(* Logix 5000 project; controller Amvex_Thorpe_Flowmeter vendor 1 type 14 code 106 rev 33.13; software revision 33.01; part 11 of 16 *)
(* tags used below, declared in another part *)
   Auto_Seq : SEQ;
   Manual_ONS : BOOL;
   Manual_Output_Reset : BOOL;
   MODE : MODE;
   RESET : BOOL;
   temp_Gripper_Delay : TIMER;
   Test : Connect;
   Air_Pressure_Issue_Delay_TMR : TIMER;
   Close : BOOL;
   Close_Rapid : Servo_Move;
   Close_Step : Servo_Move;
   Datalogging_Time_Delay : TIMER;
   HMI : HMI_Temp;
   MCP : MCP;
   MCP_00 : UDT_ID86;
   Open : BOOL;
   Reject : BOOL;
   Reject_Active : BOOL;
   Reject_Pallet_Bit : DINT;
   Test2_Step : Servo_Move;
   Test4_Step : Servo_Move;
   Test5_Step : Servo_Move;
   Test_Data : REAL[8];
   Test_Data_ONS : BOOL[32];
   Test_Delay_TMR : TIMER[5];
   Transmit_Data : BOOL;
   Vision_Result_OK_TMR : TIMER[6];
   Vision_TMR : TIMER[3];
(* MCP_Main, continued *)

ROUTINE NEW_YEAR   (* ladder *)
END_ROUTINE

ROUTINE R01_INPUTS   (* ladder *)
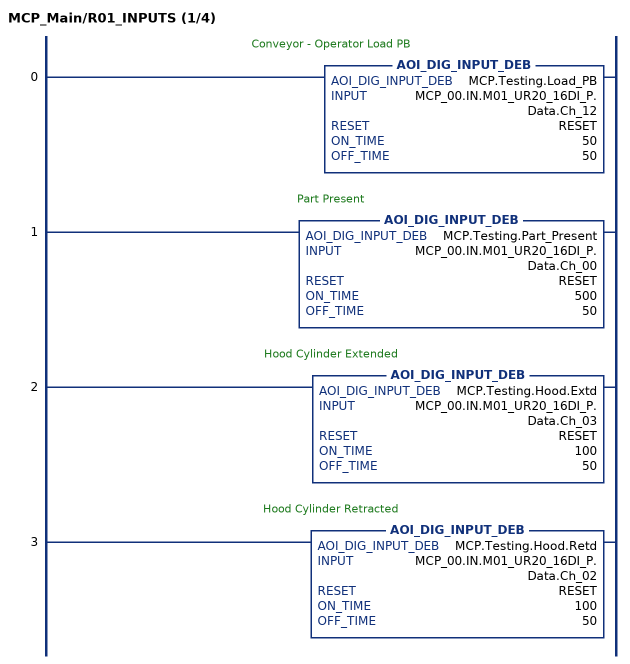
   // Conveyor - Operator Load PB
   0: AOI_DIG_INPUT_DEB(MCP.Testing.Load_PB,MCP_00.IN.M01_UR20_16DI_P.Data.Ch_12,RESET,50,50);
   // Part Present
   1: AOI_DIG_INPUT_DEB(MCP.Testing.Part_Present,MCP_00.IN.M01_UR20_16DI_P.Data.Ch_00,RESET,500,50);
   // Hood Cylinder Extended
   2: AOI_DIG_INPUT_DEB(MCP.Testing.Hood.Extd,MCP_00.IN.M01_UR20_16DI_P.Data.Ch_03,RESET,100,50);
   // Hood Cylinder Retracted
   3: AOI_DIG_INPUT_DEB(MCP.Testing.Hood.Retd,MCP_00.IN.M01_UR20_16DI_P.Data.Ch_02,RESET,100,50);
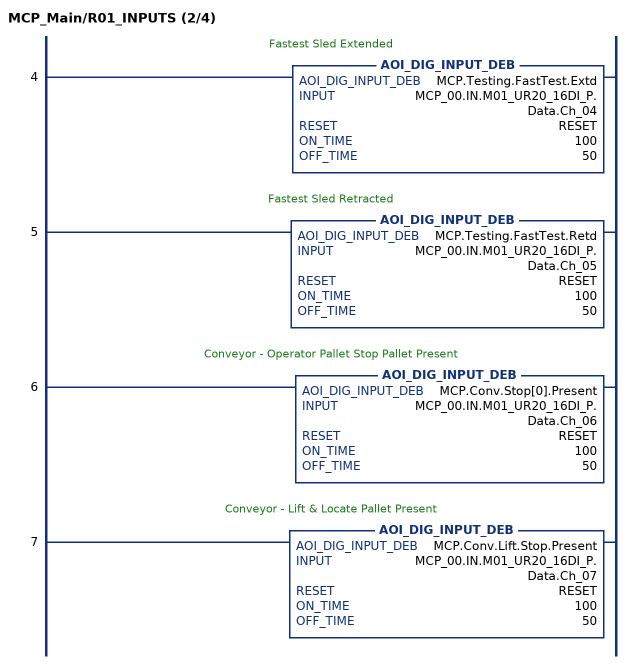
   // Fastest Sled Extended
   4: AOI_DIG_INPUT_DEB(MCP.Testing.FastTest.Extd,MCP_00.IN.M01_UR20_16DI_P.Data.Ch_04,RESET,100,50);
   // Fastest Sled Retracted
   5: AOI_DIG_INPUT_DEB(MCP.Testing.FastTest.Retd,MCP_00.IN.M01_UR20_16DI_P.Data.Ch_05,RESET,100,50);
   // Conveyor - Operator Pallet Stop Pallet Present
   6: AOI_DIG_INPUT_DEB(MCP.Conv.Stop[0].Present,MCP_00.IN.M01_UR20_16DI_P.Data.Ch_06,RESET,100,50);
   // Conveyor - Lift & Locate Pallet Present
   7: AOI_DIG_INPUT_DEB(MCP.Conv.Lift.Stop.Present,MCP_00.IN.M01_UR20_16DI_P.Data.Ch_07,RESET,100,50);
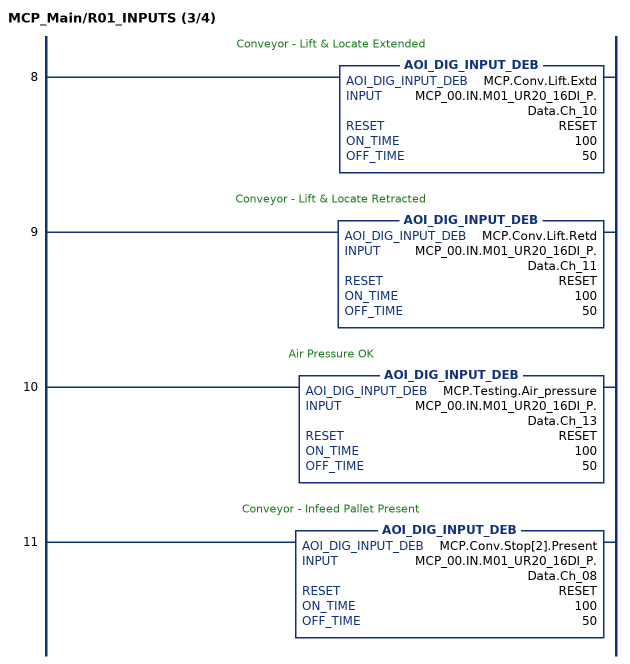
   // Conveyor - Lift & Locate Extended
   8: AOI_DIG_INPUT_DEB(MCP.Conv.Lift.Extd,MCP_00.IN.M01_UR20_16DI_P.Data.Ch_10,RESET,100,50);
   // Conveyor - Lift & Locate Retracted
   9: AOI_DIG_INPUT_DEB(MCP.Conv.Lift.Retd,MCP_00.IN.M01_UR20_16DI_P.Data.Ch_11,RESET,100,50);
   // Air Pressure OK
   10: AOI_DIG_INPUT_DEB(MCP.Testing.Air_pressure,MCP_00.IN.M01_UR20_16DI_P.Data.Ch_13,RESET,100,50);
   // Conveyor - Infeed Pallet Present
   11: AOI_DIG_INPUT_DEB(MCP.Conv.Stop[2].Present,MCP_00.IN.M01_UR20_16DI_P.Data.Ch_08,RESET,100,50);
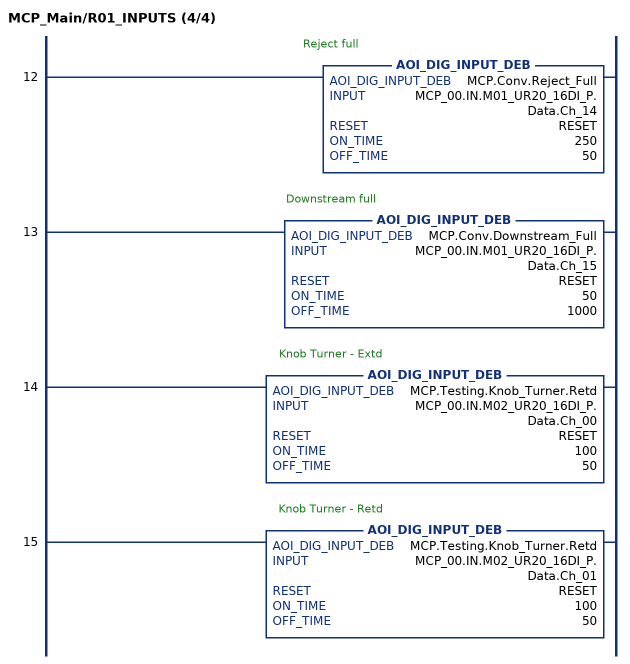
   // Reject full
   12: AOI_DIG_INPUT_DEB(MCP.Conv.Reject_Full,MCP_00.IN.M01_UR20_16DI_P.Data.Ch_14,RESET,250,50);
   // Downstream full
   13: AOI_DIG_INPUT_DEB(MCP.Conv.Downstream_Full,MCP_00.IN.M01_UR20_16DI_P.Data.Ch_15,RESET,50,1000);
   // Knob Turner - Extd
   14: AOI_DIG_INPUT_DEB(MCP.Testing.Knob_Turner.Retd,MCP_00.IN.M02_UR20_16DI_P.Data.Ch_00,RESET,100,50);
   // Knob Turner - Retd
   15: AOI_DIG_INPUT_DEB(MCP.Testing.Knob_Turner.Retd,MCP_00.IN.M02_UR20_16DI_P.Data.Ch_01,RESET,100,50);
END_ROUTINE

ROUTINE R02_OUTPUTS   (* ladder *)
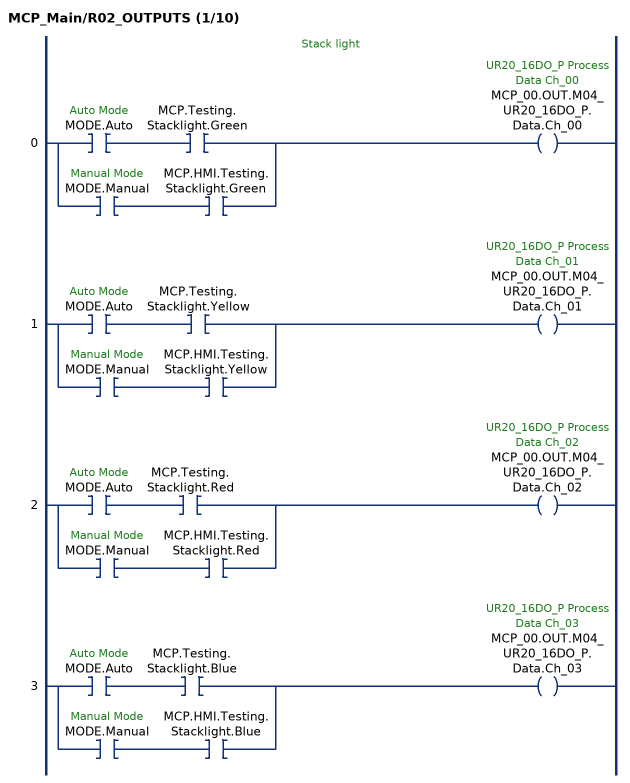
   // Stack light
   0: [XIC(MODE.Auto) XIC(MCP.Testing.Stacklight.Green) ,XIC(MODE.Manual) XIC(MCP.HMI.Testing.Stacklight.Green) ]OTE(MCP_00.OUT.M04_UR20_16DO_P.Data.Ch_00);
   1: [XIC(MODE.Auto) XIC(MCP.Testing.Stacklight.Yellow) ,XIC(MODE.Manual) XIC(MCP.HMI.Testing.Stacklight.Yellow) ]OTE(MCP_00.OUT.M04_UR20_16DO_P.Data.Ch_01);
   2: [XIC(MODE.Auto) XIC(MCP.Testing.Stacklight.Red) ,XIC(MODE.Manual) XIC(MCP.HMI.Testing.Stacklight.Red) ]OTE(MCP_00.OUT.M04_UR20_16DO_P.Data.Ch_02);
   3: [XIC(MODE.Auto) XIC(MCP.Testing.Stacklight.Blue) ,XIC(MODE.Manual) XIC(MCP.HMI.Testing.Stacklight.Blue) ]OTE(MCP_00.OUT.M04_UR20_16DO_P.Data.Ch_03);
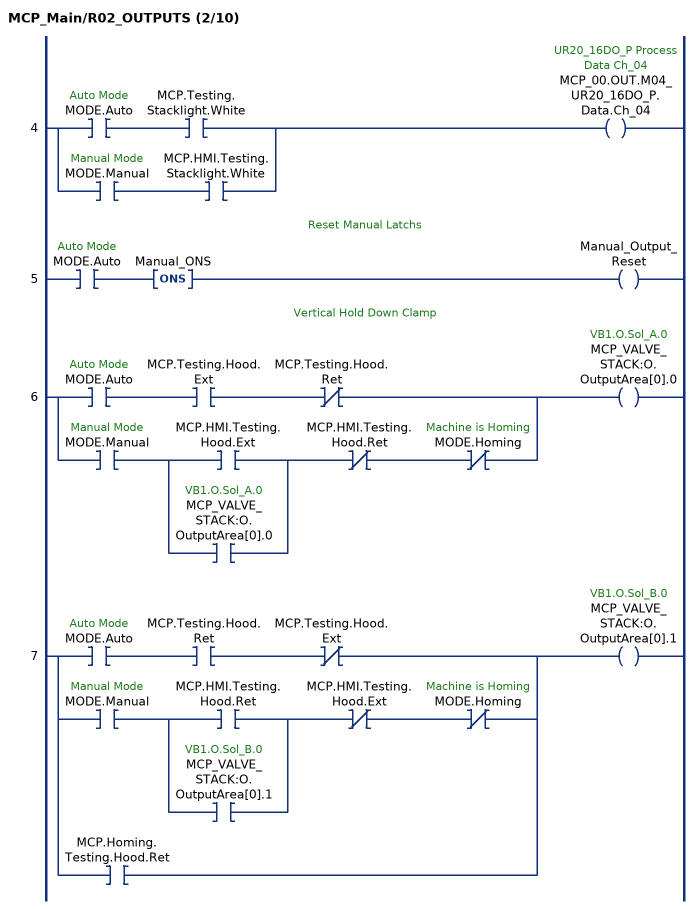
   4: [XIC(MODE.Auto) XIC(MCP.Testing.Stacklight.White) ,XIC(MODE.Manual) XIC(MCP.HMI.Testing.Stacklight.White) ]OTE(MCP_00.OUT.M04_UR20_16DO_P.Data.Ch_04);
   // Reset Manual Latchs
   5: XIC(MODE.Auto)ONS(Manual_ONS)OTE(Manual_Output_Reset);
   // Vertical Hold Down Clamp
   6: [XIC(MODE.Auto) XIC(MCP.Testing.Hood.Ext) XIO(MCP.Testing.Hood.Ret) ,XIC(MODE.Manual) [XIC(MCP.HMI.Testing.Hood.Ext) ,XIC(MCP_VALVE_STACK:O.OutputArea[0].0) ] XIO(MCP.HMI.Testing.Hood.Ret) XIO(MODE.Homing) ]OTE(MCP_VALVE_STACK:O.OutputArea[0].0);
   7: [XIC(MODE.Auto) XIC(MCP.Testing.Hood.Ret) XIO(MCP.Testing.Hood.Ext) ,XIC(MODE.Manual) [XIC(MCP.HMI.Testing.Hood.Ret) ,XIC(MCP_VALVE_STACK:O.OutputArea[0].1) ] XIO(MCP.HMI.Testing.Hood.Ext) XIO(MODE.Homing) ,XIC(MCP.Homing.Testing.Hood.Ret) ]OTE(MCP_VALVE_STACK:O.OutputArea[0].1);
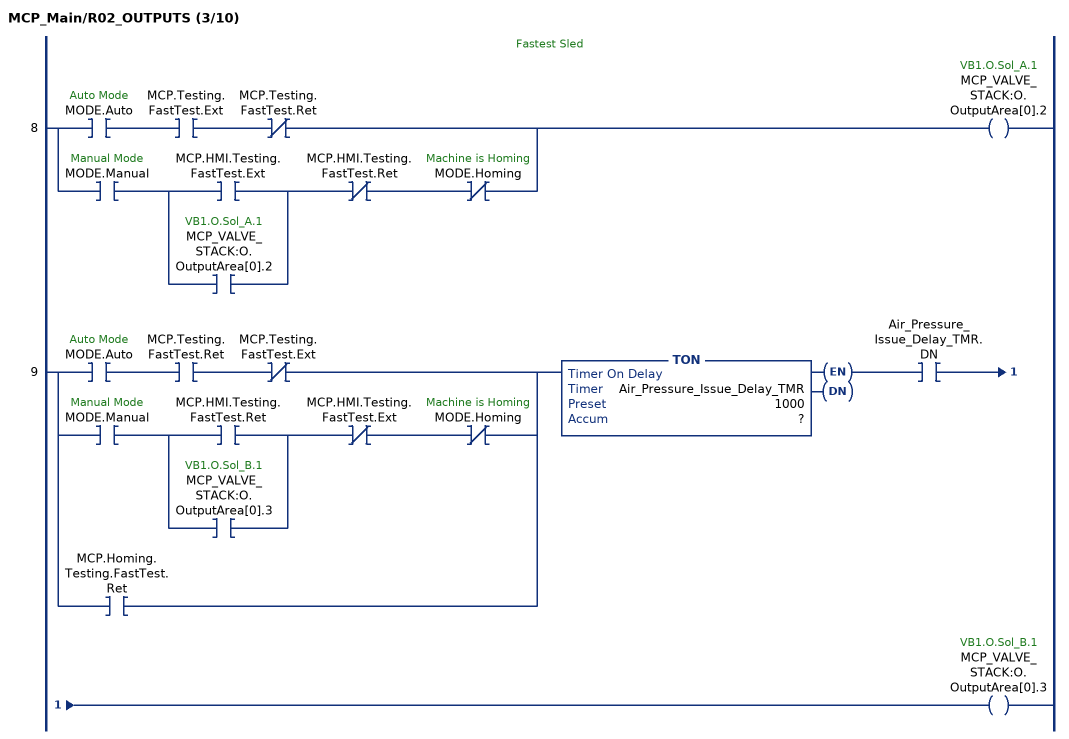
   // Fastest Sled
   8: [XIC(MODE.Auto) XIC(MCP.Testing.FastTest.Ext) XIO(MCP.Testing.FastTest.Ret) ,XIC(MODE.Manual) [XIC(MCP.HMI.Testing.FastTest.Ext) ,XIC(MCP_VALVE_STACK:O.OutputArea[0].2) ] XIO(MCP.HMI.Testing.FastTest.Ret) XIO(MODE.Homing) ]OTE(MCP_VALVE_STACK:O.OutputArea[0].2);
   9: [XIC(MODE.Auto) XIC(MCP.Testing.FastTest.Ret) XIO(MCP.Testing.FastTest.Ext) ,XIC(MODE.Manual) [XIC(MCP.HMI.Testing.FastTest.Ret) ,XIC(MCP_VALVE_STACK:O.OutputArea[0].3) ] XIO(MCP.HMI.Testing.FastTest.Ext) XIO(MODE.Homing) ,XIC(MCP.Homing.Testing.FastTest.Ret) ]TON(Air_Pressure_Issue_Delay_TMR,?,?)XIC(Air_Pressure_Issue_Delay_TMR.DN)OTE(MCP_VALVE_STACK:O.OutputArea[0].3);
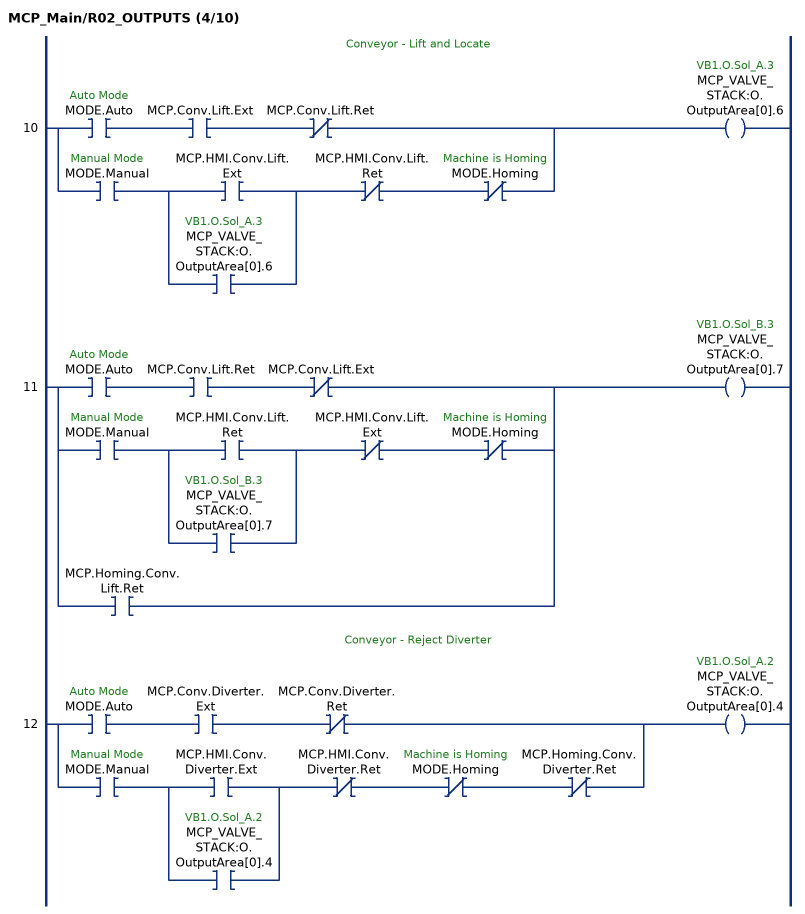
   // Conveyor - Lift and Locate
   10: [XIC(MODE.Auto) XIC(MCP.Conv.Lift.Ext) XIO(MCP.Conv.Lift.Ret) ,XIC(MODE.Manual) [XIC(MCP.HMI.Conv.Lift.Ext) ,XIC(MCP_VALVE_STACK:O.OutputArea[0].6) ] XIO(MCP.HMI.Conv.Lift.Ret) XIO(MODE.Homing) ]OTE(MCP_VALVE_STACK:O.OutputArea[0].6);
   11: [XIC(MODE.Auto) XIC(MCP.Conv.Lift.Ret) XIO(MCP.Conv.Lift.Ext) ,XIC(MODE.Manual) [XIC(MCP.HMI.Conv.Lift.Ret) ,XIC(MCP_VALVE_STACK:O.OutputArea[0].7) ] XIO(MCP.HMI.Conv.Lift.Ext) XIO(MODE.Homing) ,XIC(MCP.Homing.Conv.Lift.Ret) ]OTE(MCP_VALVE_STACK:O.OutputArea[0].7);
   // Conveyor - Reject Diverter
   12: [XIC(MODE.Auto) XIC(MCP.Conv.Diverter.Ext) XIO(MCP.Conv.Diverter.Ret) ,XIC(MODE.Manual) [XIC(MCP.HMI.Conv.Diverter.Ext) ,XIC(MCP_VALVE_STACK:O.OutputArea[0].4) ] XIO(MCP.HMI.Conv.Diverter.Ret) XIO(MODE.Homing) XIO(MCP.Homing.Conv.Diverter.Ret) ]OTE(MCP_VALVE_STACK:O.OutputArea[0].4);
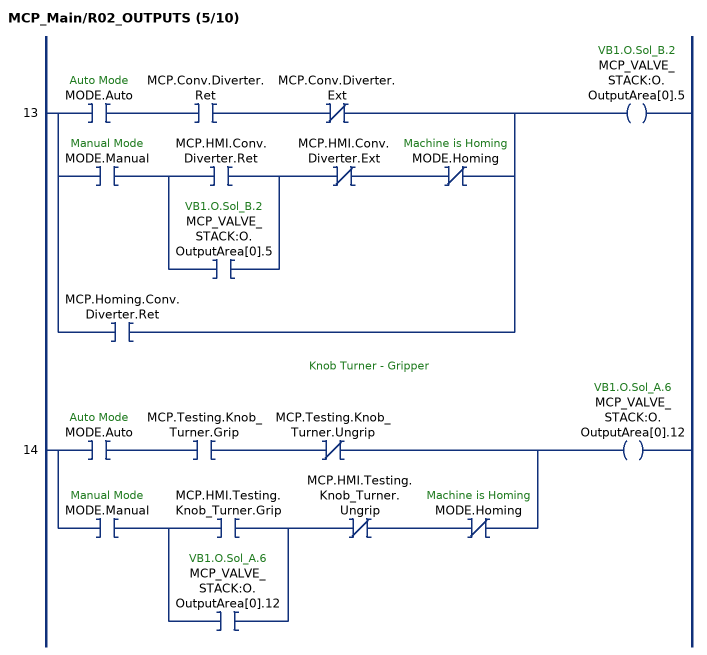
   13: [XIC(MODE.Auto) XIC(MCP.Conv.Diverter.Ret) XIO(MCP.Conv.Diverter.Ext) ,XIC(MODE.Manual) [XIC(MCP.HMI.Conv.Diverter.Ret) ,XIC(MCP_VALVE_STACK:O.OutputArea[0].5) ] XIO(MCP.HMI.Conv.Diverter.Ext) XIO(MODE.Homing) ,XIC(MCP.Homing.Conv.Diverter.Ret) ]OTE(MCP_VALVE_STACK:O.OutputArea[0].5);
   // Knob Turner - Gripper
   14: [XIC(MODE.Auto) XIC(MCP.Testing.Knob_Turner.Grip) XIO(MCP.Testing.Knob_Turner.Ungrip) ,XIC(MODE.Manual) [XIC(MCP.HMI.Testing.Knob_Turner.Grip) ,XIC(MCP_VALVE_STACK:O.OutputArea[0].12) ] XIO(MCP.HMI.Testing.Knob_Turner.Ungrip) XIO(MODE.Homing) ]OTE(MCP_VALVE_STACK:O.OutputArea[0].12);
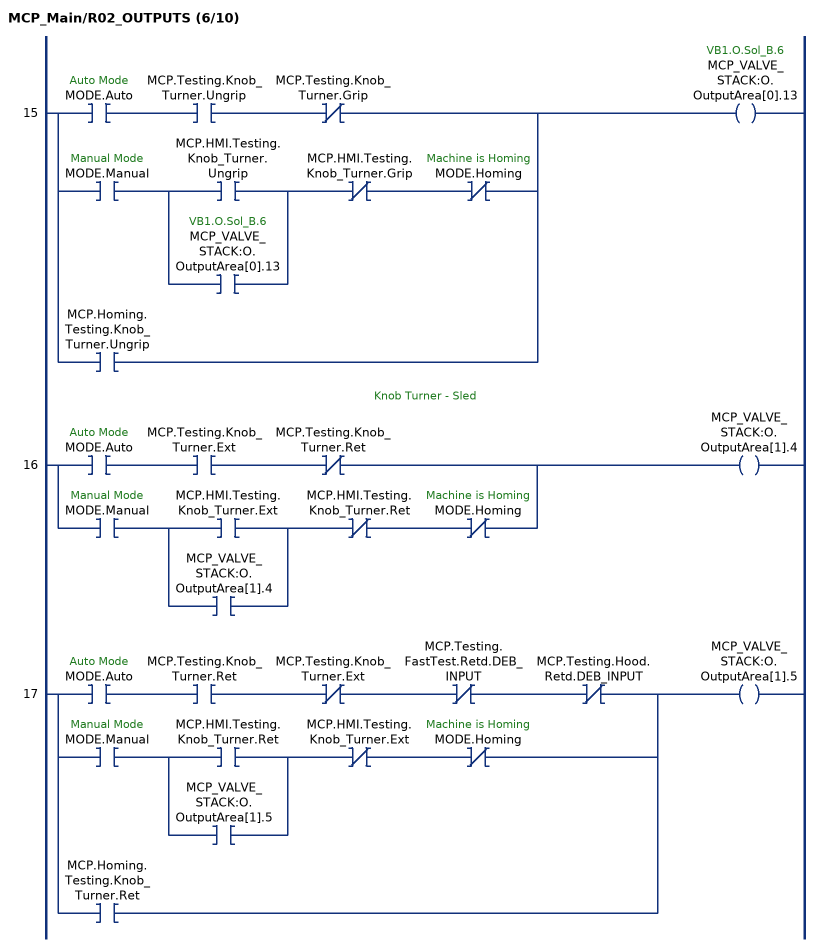
   15: [XIC(MODE.Auto) XIC(MCP.Testing.Knob_Turner.Ungrip) XIO(MCP.Testing.Knob_Turner.Grip) ,XIC(MODE.Manual) [XIC(MCP.HMI.Testing.Knob_Turner.Ungrip) ,XIC(MCP_VALVE_STACK:O.OutputArea[0].13) ] XIO(MCP.HMI.Testing.Knob_Turner.Grip) XIO(MODE.Homing) ,XIC(MCP.Homing.Testing.Knob_Turner.Ungrip) ]OTE(MCP_VALVE_STACK:O.OutputArea[0].13);
   // Knob Turner - Sled
   16: [XIC(MODE.Auto) XIC(MCP.Testing.Knob_Turner.Ext) XIO(MCP.Testing.Knob_Turner.Ret) ,XIC(MODE.Manual) [XIC(MCP.HMI.Testing.Knob_Turner.Ext) ,XIC(MCP_VALVE_STACK:O.OutputArea[1].4) ] XIO(MCP.HMI.Testing.Knob_Turner.Ret) XIO(MODE.Homing) ]OTE(MCP_VALVE_STACK:O.OutputArea[1].4);
   17: [XIC(MODE.Auto) XIC(MCP.Testing.Knob_Turner.Ret) XIO(MCP.Testing.Knob_Turner.Ext) XIO(MCP.Testing.FastTest.Retd.DEB_INPUT) XIO(MCP.Testing.Hood.Retd.DEB_INPUT) ,XIC(MODE.Manual) [XIC(MCP.HMI.Testing.Knob_Turner.Ret) ,XIC(MCP_VALVE_STACK:O.OutputArea[1].5) ] XIO(MCP.HMI.Testing.Knob_Turner.Ext) XIO(MODE.Homing) ,XIC(MCP.Homing.Testing.Knob_Turner.Ret) ]OTE(MCP_VALVE_STACK:O.OutputArea[1].5);
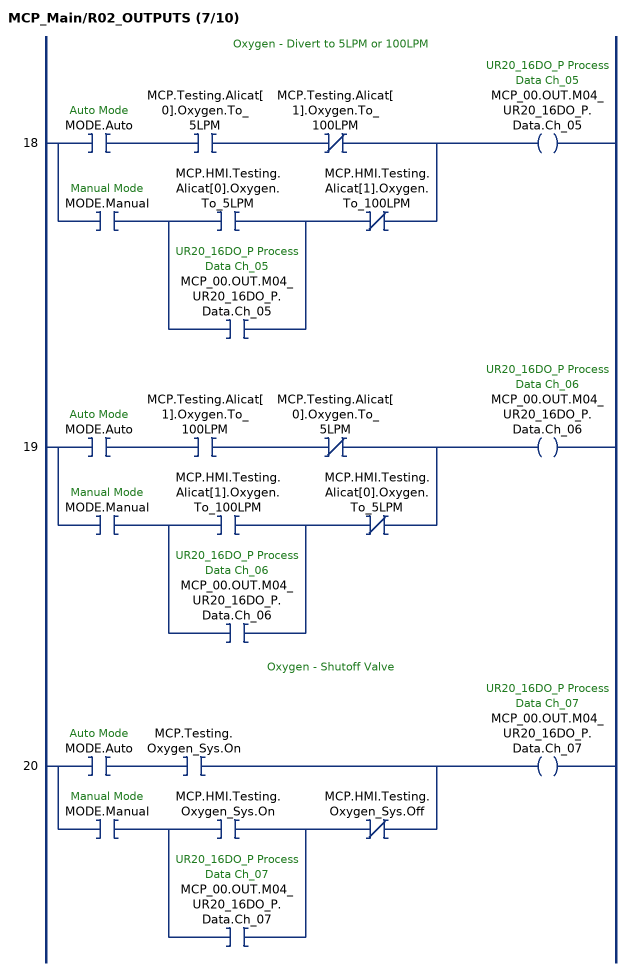
   // Oxygen - Divert to 5LPM or 100LPM
   18: [XIC(MODE.Auto) XIC(MCP.Testing.Alicat[0].Oxygen.To_5LPM) XIO(MCP.Testing.Alicat[1].Oxygen.To_100LPM) ,XIC(MODE.Manual) [XIC(MCP.HMI.Testing.Alicat[0].Oxygen.To_5LPM) ,XIC(MCP_00.OUT.M04_UR20_16DO_P.Data.Ch_05) ] XIO(MCP.HMI.Testing.Alicat[1].Oxygen.To_100LPM) ]OTE(MCP_00.OUT.M04_UR20_16DO_P.Data.Ch_05);
   19: [XIC(MODE.Auto) XIC(MCP.Testing.Alicat[1].Oxygen.To_100LPM) XIO(MCP.Testing.Alicat[0].Oxygen.To_5LPM) ,XIC(MODE.Manual) [XIC(MCP.HMI.Testing.Alicat[1].Oxygen.To_100LPM) ,XIC(MCP_00.OUT.M04_UR20_16DO_P.Data.Ch_06) ] XIO(MCP.HMI.Testing.Alicat[0].Oxygen.To_5LPM) ]OTE(MCP_00.OUT.M04_UR20_16DO_P.Data.Ch_06);
   // Oxygen - Shutoff Valve
   20: [XIC(MODE.Auto) XIC(MCP.Testing.Oxygen_Sys.On) ,XIC(MODE.Manual) [XIC(MCP.HMI.Testing.Oxygen_Sys.On) ,XIC(MCP_00.OUT.M04_UR20_16DO_P.Data.Ch_07) ] XIO(MCP.HMI.Testing.Oxygen_Sys.Off) ]OTE(MCP_00.OUT.M04_UR20_16DO_P.Data.Ch_07);
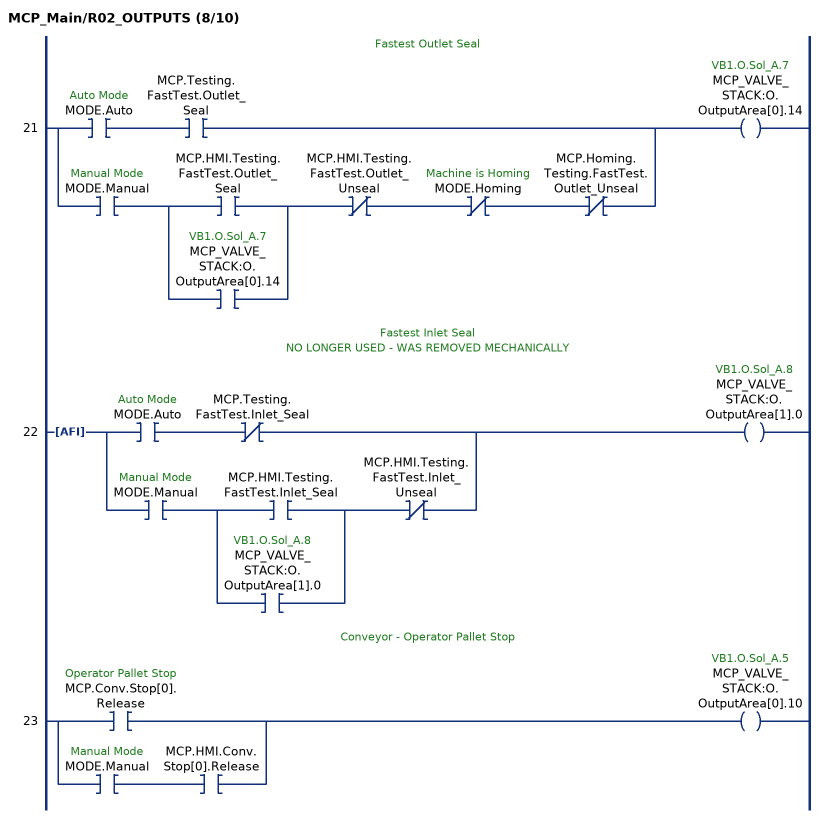
   // Fastest Outlet Seal
   21: [XIC(MODE.Auto) XIC(MCP.Testing.FastTest.Outlet_Seal) ,XIC(MODE.Manual) [XIC(MCP.HMI.Testing.FastTest.Outlet_Seal) ,XIC(MCP_VALVE_STACK:O.OutputArea[0].14) ] XIO(MCP.HMI.Testing.FastTest.Outlet_Unseal) XIO(MODE.Homing) XIO(MCP.Homing.Testing.FastTest.Outlet_Unseal) ]OTE(MCP_VALVE_STACK:O.OutputArea[0].14);
   // Fastest Inlet Seal
   // NO LONGER USED - WAS REMOVED MECHANICALLY
   22: AFI()[XIC(MODE.Auto) XIO(MCP.Testing.FastTest.Inlet_Seal) ,XIC(MODE.Manual) [XIC(MCP.HMI.Testing.FastTest.Inlet_Seal) ,XIC(MCP_VALVE_STACK:O.OutputArea[1].0) ] XIO(MCP.HMI.Testing.FastTest.Inlet_Unseal) ]OTE(MCP_VALVE_STACK:O.OutputArea[1].0);
   // Conveyor - Operator Pallet Stop
   23: [XIC(MCP.Conv.Stop[0].Release) ,XIC(MODE.Manual) XIC(MCP.HMI.Conv.Stop[0].Release) ]OTE(MCP_VALVE_STACK:O.OutputArea[0].10);
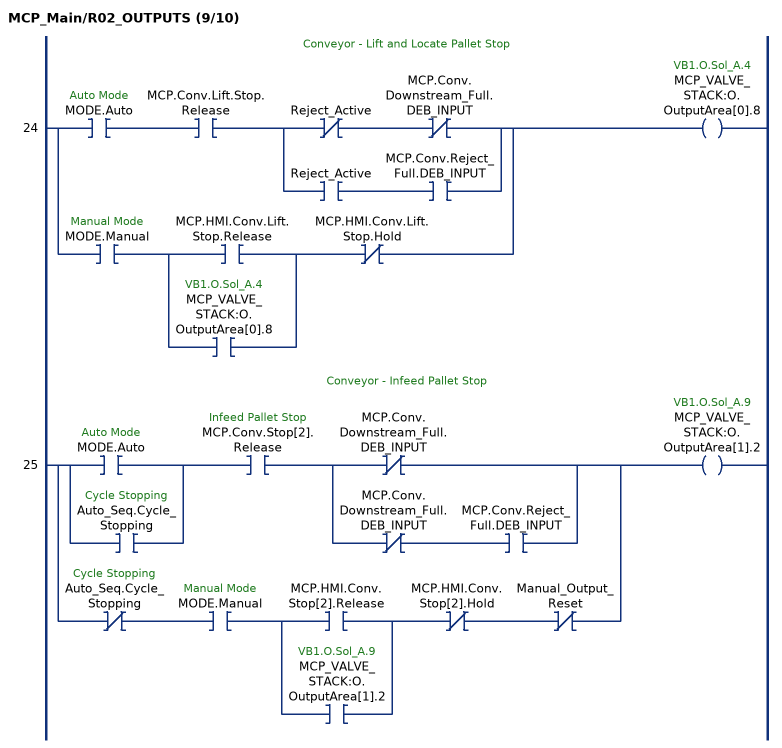
   // Conveyor - Lift and Locate Pallet Stop
   24: [XIC(MODE.Auto) XIC(MCP.Conv.Lift.Stop.Release) [XIO(Reject_Active) XIO(MCP.Conv.Downstream_Full.DEB_INPUT) ,XIC(Reject_Active) XIC(MCP.Conv.Reject_Full.DEB_INPUT) ] ,XIC(MODE.Manual) [XIC(MCP.HMI.Conv.Lift.Stop.Release) ,XIC(MCP_VALVE_STACK:O.OutputArea[0].8) ] XIO(MCP.HMI.Conv.Lift.Stop.Hold) ]OTE(MCP_VALVE_STACK:O.OutputArea[0].8);
   // Conveyor - Infeed Pallet Stop
   25: [[XIC(MODE.Auto) ,XIC(Auto_Seq.Cycle_Stopping) ] XIC(MCP.Conv.Stop[2].Release) [XIO(MCP.Conv.Downstream_Full.DEB_INPUT) ,XIO(MCP.Conv.Downstream_Full.DEB_INPUT) XIC(MCP.Conv.Reject_Full.DEB_INPUT) ] ,XIO(Auto_Seq.Cycle_Stopping) XIC(MODE.Manual) [XIC(MCP.HMI.Conv.Stop[2].Release) ,XIC(MCP_VALVE_STACK:O.OutputArea[1].2) ] XIO(MCP.HMI.Conv.Stop[2].Hold) XIO(Manual_Output_Reset) ]OTE(MCP_VALVE_STACK:O.OutputArea[1].2);
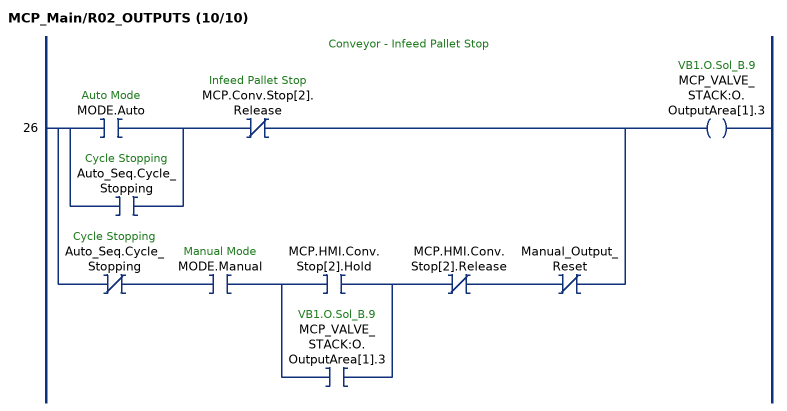
   // Conveyor - Infeed Pallet Stop
   26: [[XIC(MODE.Auto) ,XIC(Auto_Seq.Cycle_Stopping) ] XIO(MCP.Conv.Stop[2].Release) ,XIO(Auto_Seq.Cycle_Stopping) XIC(MODE.Manual) [XIC(MCP.HMI.Conv.Stop[2].Hold) ,XIC(MCP_VALVE_STACK:O.OutputArea[1].3) ] XIO(MCP.HMI.Conv.Stop[2].Release) XIO(Manual_Output_Reset) ]OTE(MCP_VALVE_STACK:O.OutputArea[1].3);
END_ROUTINE

ROUTINE R03_AUTO_SEQ   (* ladder *)
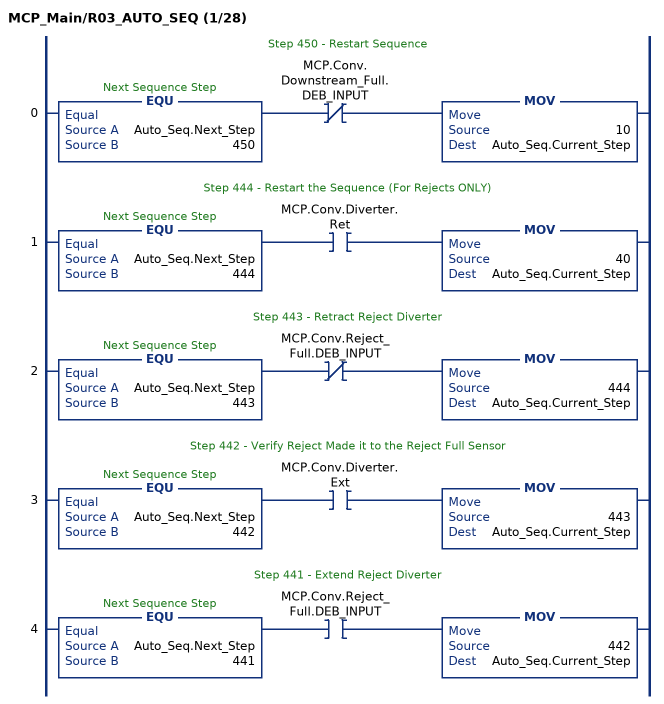
   // Step 450 - Restart Sequence
   0: EQU(Auto_Seq.Next_Step,450)XIO(MCP.Conv.Downstream_Full.DEB_INPUT)MOV(10,Auto_Seq.Current_Step);
   // Step 444 - Restart the Sequence (For Rejects ONLY)
   1: EQU(Auto_Seq.Next_Step,444)XIC(MCP.Conv.Diverter.Ret)MOV(40,Auto_Seq.Current_Step);
   // Step 443 - Retract Reject Diverter
   2: EQU(Auto_Seq.Next_Step,443)XIO(MCP.Conv.Reject_Full.DEB_INPUT)MOV(444,Auto_Seq.Current_Step);
   // Step 442 - Verify Reject Made it to the Reject Full Sensor
   3: EQU(Auto_Seq.Next_Step,442)XIC(MCP.Conv.Diverter.Ext)MOV(443,Auto_Seq.Current_Step);
   // Step 441 - Extend Reject Diverter
   4: EQU(Auto_Seq.Next_Step,441)XIC(MCP.Conv.Reject_Full.DEB_INPUT)MOV(442,Auto_Seq.Current_Step);
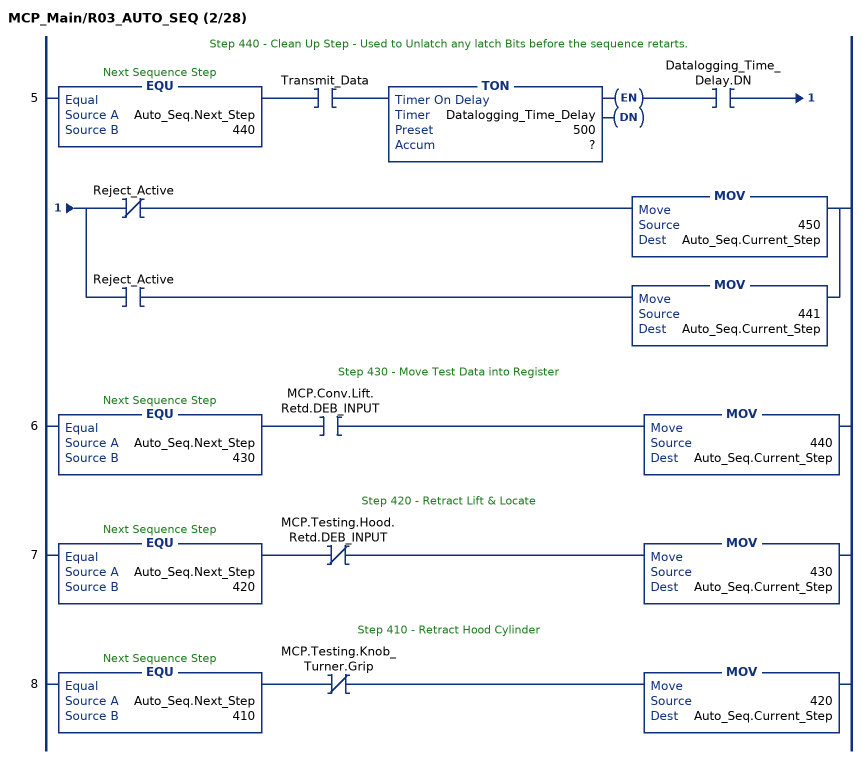
   // Step 440 - Clean Up Step - Used to Unlatch any latch Bits before the sequence retarts.
   5: EQU(Auto_Seq.Next_Step,440)XIC(Transmit_Data)TON(Datalogging_Time_Delay,?,?)XIC(Datalogging_Time_Delay.DN)[XIO(Reject_Active) MOV(450,Auto_Seq.Current_Step) ,XIC(Reject_Active) MOV(441,Auto_Seq.Current_Step) ];
   // Step 430 - Move Test Data into Register
   6: EQU(Auto_Seq.Next_Step,430)XIC(MCP.Conv.Lift.Retd.DEB_INPUT)MOV(440,Auto_Seq.Current_Step);
   // Step 420 - Retract Lift & Locate
   7: EQU(Auto_Seq.Next_Step,420)XIO(MCP.Testing.Hood.Retd.DEB_INPUT)MOV(430,Auto_Seq.Current_Step);
   // Step 410 - Retract Hood Cylinder
   8: EQU(Auto_Seq.Next_Step,410)XIO(MCP.Testing.Knob_Turner.Grip)MOV(420,Auto_Seq.Current_Step);
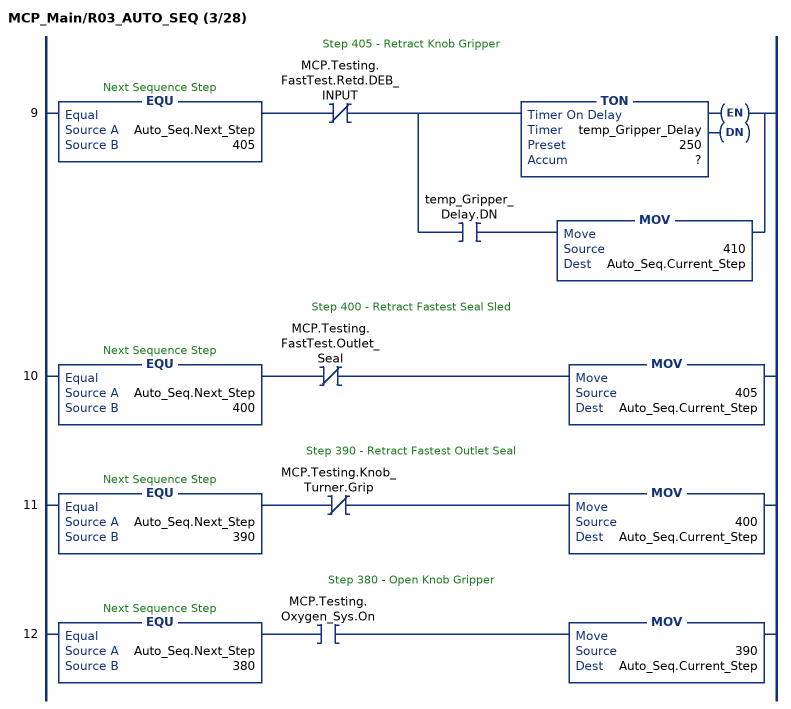
   // Step 405 - Retract Knob Gripper
   9: EQU(Auto_Seq.Next_Step,405)XIO(MCP.Testing.FastTest.Retd.DEB_INPUT)[TON(temp_Gripper_Delay,?,?) ,XIC(temp_Gripper_Delay.DN) MOV(410,Auto_Seq.Current_Step) ];
   // Step 400 - Retract Fastest Seal Sled
   10: EQU(Auto_Seq.Next_Step,400)XIO(MCP.Testing.FastTest.Outlet_Seal)MOV(405,Auto_Seq.Current_Step);
   // Step 390 - Retract Fastest Outlet Seal
   11: EQU(Auto_Seq.Next_Step,390)XIO(MCP.Testing.Knob_Turner.Grip)MOV(400,Auto_Seq.Current_Step);
   // Step 380 - Open Knob Gripper
   12: EQU(Auto_Seq.Next_Step,380)XIC(MCP.Testing.Oxygen_Sys.On)MOV(390,Auto_Seq.Current_Step);
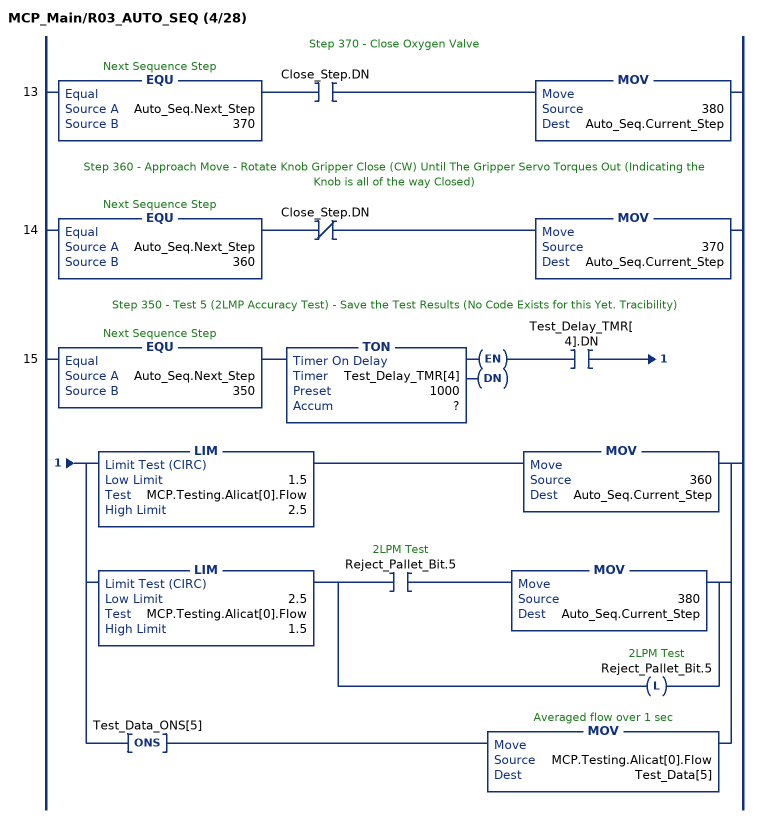
   // Step 370 - Close Oxygen Valve
   13: EQU(Auto_Seq.Next_Step,370)XIC(Close_Step.DN)MOV(380,Auto_Seq.Current_Step);
   // Step 360 - Approach Move - Rotate Knob Gripper Close (CW) Until The Gripper Servo Torques Out (Indicating the Knob is all of the way Closed)
   14: EQU(Auto_Seq.Next_Step,360)XIO(Close_Step.DN)MOV(370,Auto_Seq.Current_Step);
   // Step 350 - Test 5 (2LMP Accuracy Test) - Save the Test Results (No Code Exists for this Yet. Tracibility)
   15: EQU(Auto_Seq.Next_Step,350)TON(Test_Delay_TMR[4],?,?)XIC(Test_Delay_TMR[4].DN)[LIM(1.5,MCP.Testing.Alicat[0].Flow,2.5) MOV(360,Auto_Seq.Current_Step) ,LIM(2.5,MCP.Testing.Alicat[0].Flow,1.5) [XIC(Reject_Pallet_Bit.5) MOV(380,Auto_Seq.Current_Step) ,OTL(Reject_Pallet_Bit.5) ] ,ONS(Test_Data_ONS[5]) MOV(MCP.Testing.Alicat[0].Flow,Test_Data[5]) ];
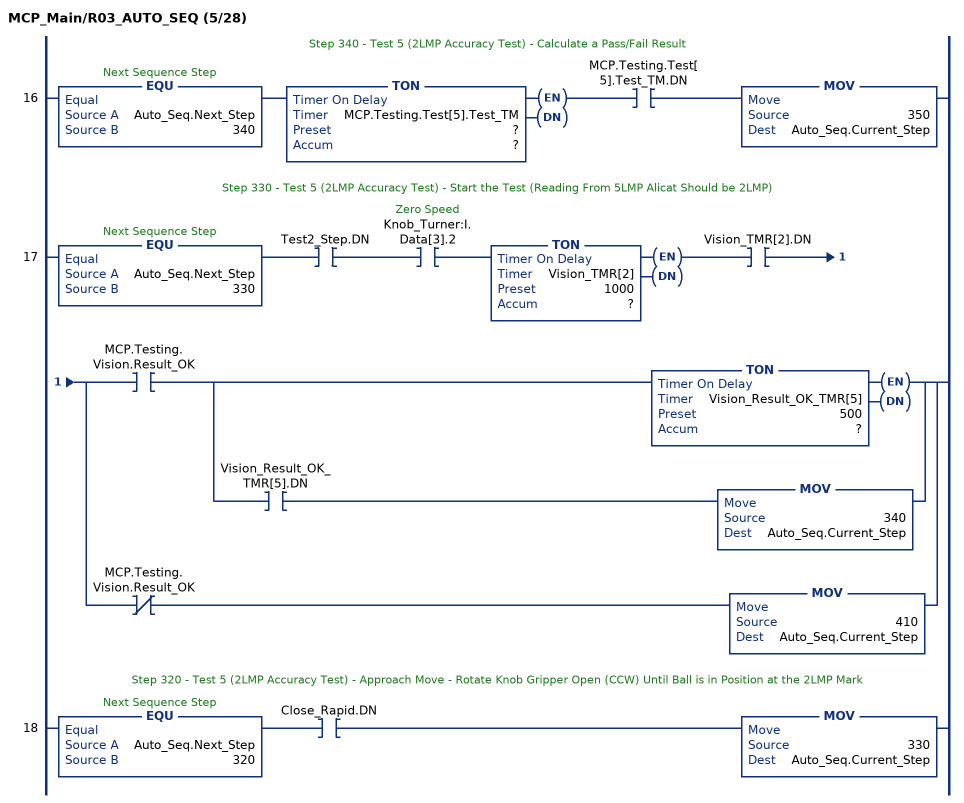
   // Step 340 - Test 5 (2LMP Accuracy Test) - Calculate a Pass/Fail Result
   16: EQU(Auto_Seq.Next_Step,340)TON(MCP.Testing.Test[5].Test_TM,?,?)XIC(MCP.Testing.Test[5].Test_TM.DN)MOV(350,Auto_Seq.Current_Step);
   // Step 330 - Test 5 (2LMP Accuracy Test) - Start the Test (Reading From 5LMP Alicat Should be 2LMP)
   17: EQU(Auto_Seq.Next_Step,330)XIC(Test2_Step.DN)XIC(Knob_Turner:I.Data[3].2)TON(Vision_TMR[2],?,?)XIC(Vision_TMR[2].DN)[XIC(MCP.Testing.Vision.Result_OK) [TON(Vision_Result_OK_TMR[5],?,?) ,XIC(Vision_Result_OK_TMR[5].DN) MOV(340,Auto_Seq.Current_Step) ] ,XIO(MCP.Testing.Vision.Result_OK) MOV(410,Auto_Seq.Current_Step) ];
   // Step 320 - Test 5 (2LMP Accuracy Test) - Approach Move - Rotate Knob Gripper Open (CCW) Until Ball is in Position at the 2LMP Mark
   18: EQU(Auto_Seq.Next_Step,320)XIC(Close_Rapid.DN)MOV(330,Auto_Seq.Current_Step);
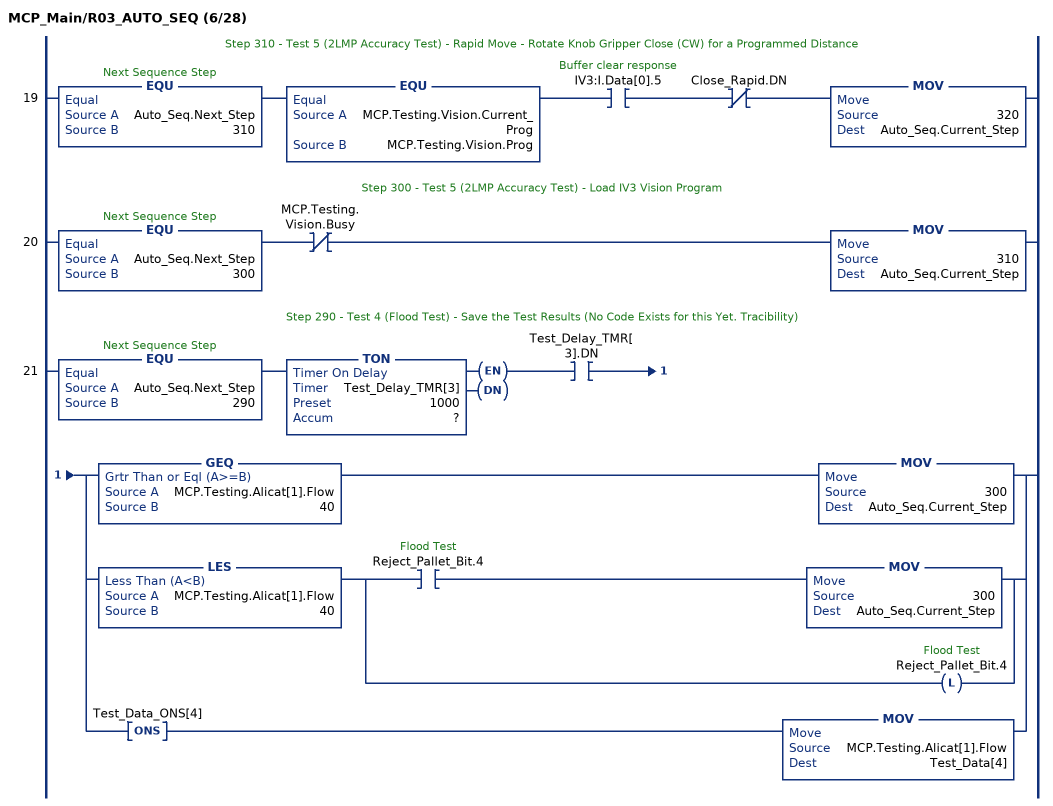
   // Step 310 - Test 5 (2LMP Accuracy Test) - Rapid Move - Rotate Knob Gripper Close (CW) for a Programmed Distance
   19: EQU(Auto_Seq.Next_Step,310)EQU(MCP.Testing.Vision.Current_Prog,MCP.Testing.Vision.Prog)XIC(IV3:I.Data[0].5)XIO(Close_Rapid.DN)MOV(320,Auto_Seq.Current_Step);
   // Step 300 - Test 5 (2LMP Accuracy Test) - Load IV3 Vision Program
   20: EQU(Auto_Seq.Next_Step,300)XIO(MCP.Testing.Vision.Busy)MOV(310,Auto_Seq.Current_Step);
   // Step 290 - Test 4 (Flood Test) - Save the Test Results (No Code Exists for this Yet. Tracibility)
   21: EQU(Auto_Seq.Next_Step,290)TON(Test_Delay_TMR[3],?,?)XIC(Test_Delay_TMR[3].DN)[GEQ(MCP.Testing.Alicat[1].Flow,40) MOV(300,Auto_Seq.Current_Step) ,LES(MCP.Testing.Alicat[1].Flow,40) [XIC(Reject_Pallet_Bit.4) MOV(300,Auto_Seq.Current_Step) ,OTL(Reject_Pallet_Bit.4) ] ,ONS(Test_Data_ONS[4]) MOV(MCP.Testing.Alicat[1].Flow,Test_Data[4]) ];
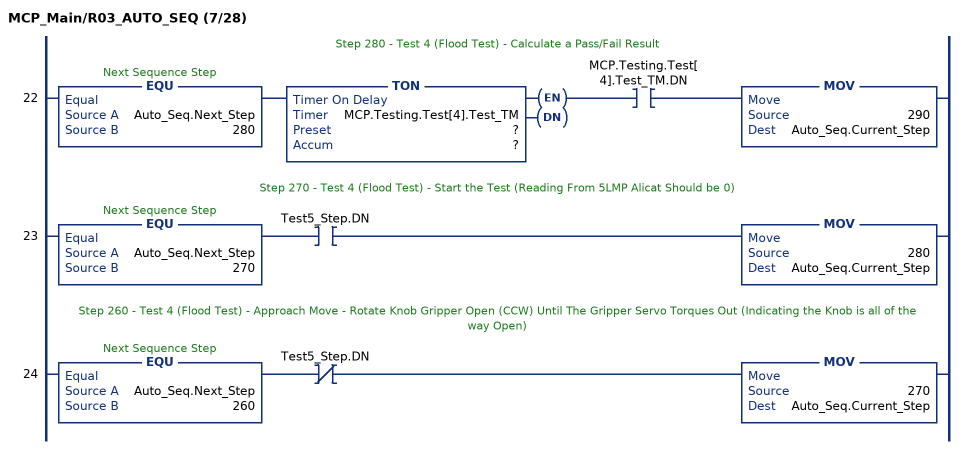
   // Step 280 - Test 4 (Flood Test) - Calculate a Pass/Fail Result
   22: EQU(Auto_Seq.Next_Step,280)TON(MCP.Testing.Test[4].Test_TM,?,?)XIC(MCP.Testing.Test[4].Test_TM.DN)MOV(290,Auto_Seq.Current_Step);
   // Step 270 - Test 4 (Flood Test) - Start the Test (Reading From 5LMP Alicat Should be 0)
   23: EQU(Auto_Seq.Next_Step,270)XIC(Test5_Step.DN)MOV(280,Auto_Seq.Current_Step);
   // Step 260 - Test 4 (Flood Test) - Approach Move - Rotate Knob Gripper Open (CCW) Until The Gripper Servo Torques Out (Indicating the Knob is all of the way Open)
   24: EQU(Auto_Seq.Next_Step,260)XIO(Test5_Step.DN)MOV(270,Auto_Seq.Current_Step);
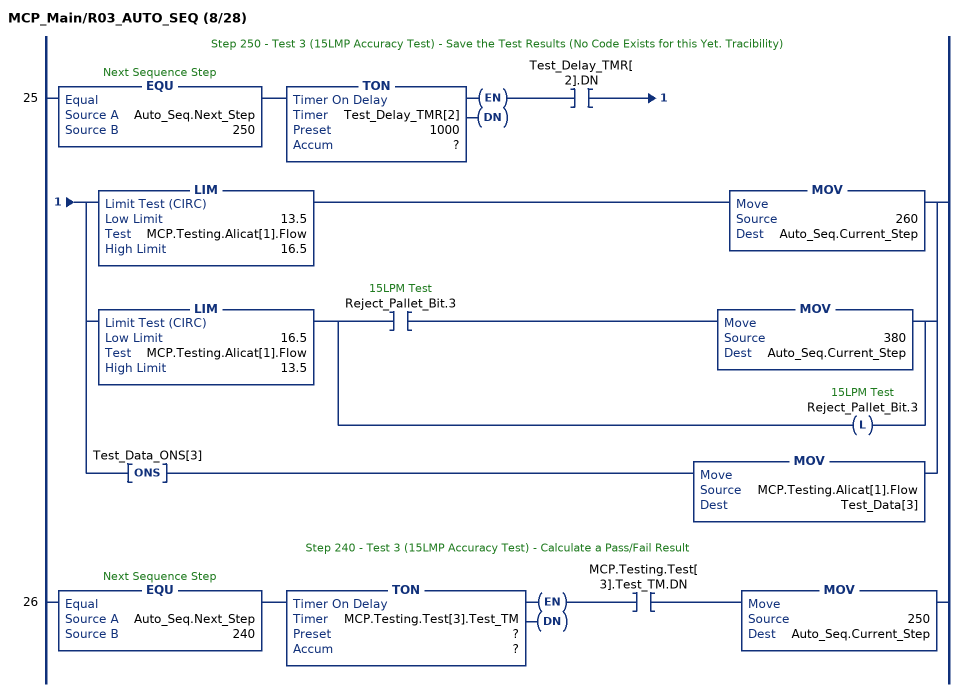
   // Step 250 - Test 3 (15LMP Accuracy Test) - Save the Test Results (No Code Exists for this Yet. Tracibility)
   25: EQU(Auto_Seq.Next_Step,250)TON(Test_Delay_TMR[2],?,?)XIC(Test_Delay_TMR[2].DN)[LIM(13.5,MCP.Testing.Alicat[1].Flow,16.5) MOV(260,Auto_Seq.Current_Step) ,LIM(16.5,MCP.Testing.Alicat[1].Flow,13.5) [XIC(Reject_Pallet_Bit.3) MOV(380,Auto_Seq.Current_Step) ,OTL(Reject_Pallet_Bit.3) ] ,ONS(Test_Data_ONS[3]) MOV(MCP.Testing.Alicat[1].Flow,Test_Data[3]) ];
   // Step 240 - Test 3 (15LMP Accuracy Test) - Calculate a Pass/Fail Result
   26: EQU(Auto_Seq.Next_Step,240)TON(MCP.Testing.Test[3].Test_TM,?,?)XIC(MCP.Testing.Test[3].Test_TM.DN)MOV(250,Auto_Seq.Current_Step);
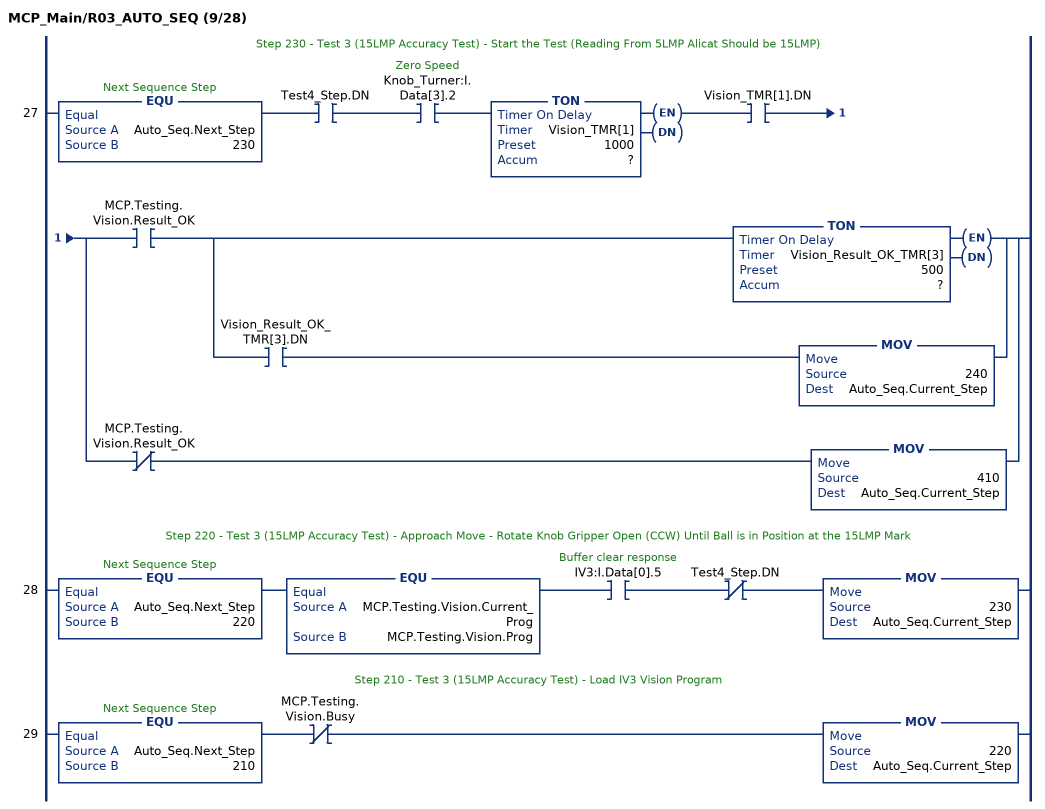
   // Step 230 - Test 3 (15LMP Accuracy Test) - Start the Test (Reading From 5LMP Alicat Should be 15LMP)
   27: EQU(Auto_Seq.Next_Step,230)XIC(Test4_Step.DN)XIC(Knob_Turner:I.Data[3].2)TON(Vision_TMR[1],?,?)XIC(Vision_TMR[1].DN)[XIC(MCP.Testing.Vision.Result_OK) [TON(Vision_Result_OK_TMR[3],?,?) ,XIC(Vision_Result_OK_TMR[3].DN) MOV(240,Auto_Seq.Current_Step) ] ,XIO(MCP.Testing.Vision.Result_OK) MOV(410,Auto_Seq.Current_Step) ];
   // Step 220 - Test 3 (15LMP Accuracy Test) - Approach Move - Rotate Knob Gripper Open (CCW) Until Ball is in Position at the 15LMP Mark
   28: EQU(Auto_Seq.Next_Step,220)EQU(MCP.Testing.Vision.Current_Prog,MCP.Testing.Vision.Prog)XIC(IV3:I.Data[0].5)XIO(Test4_Step.DN)MOV(230,Auto_Seq.Current_Step);
   // Step 210 - Test 3 (15LMP Accuracy Test) - Load IV3 Vision Program
   29: EQU(Auto_Seq.Next_Step,210)XIO(MCP.Testing.Vision.Busy)MOV(220,Auto_Seq.Current_Step);
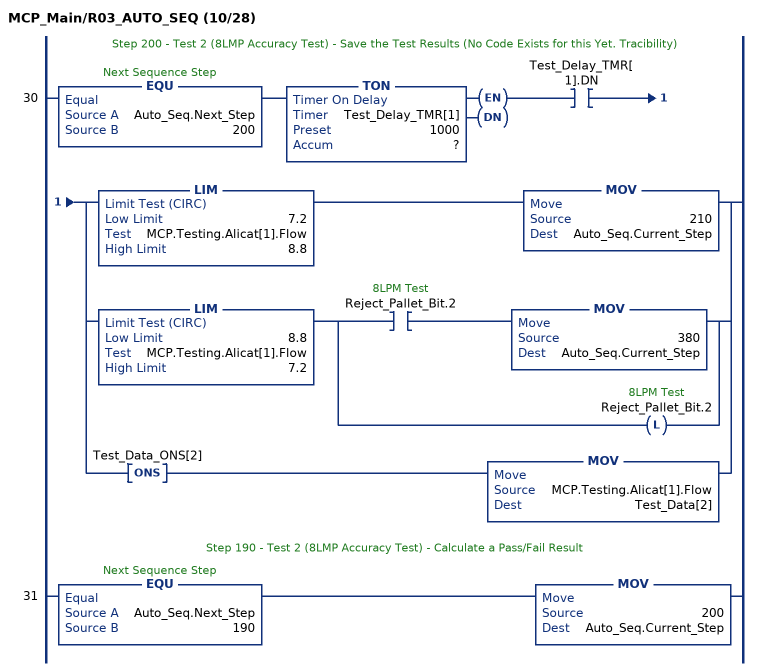
   // Step 200 - Test 2 (8LMP Accuracy Test) - Save the Test Results (No Code Exists for this Yet. Tracibility)
   30: EQU(Auto_Seq.Next_Step,200)TON(Test_Delay_TMR[1],?,?)XIC(Test_Delay_TMR[1].DN)[LIM(7.2,MCP.Testing.Alicat[1].Flow,8.8) MOV(210,Auto_Seq.Current_Step) ,LIM(8.8,MCP.Testing.Alicat[1].Flow,7.2) [XIC(Reject_Pallet_Bit.2) MOV(380,Auto_Seq.Current_Step) ,OTL(Reject_Pallet_Bit.2) ] ,ONS(Test_Data_ONS[2]) MOV(MCP.Testing.Alicat[1].Flow,Test_Data[2]) ];
   // Step 190 - Test 2 (8LMP Accuracy Test) - Calculate a Pass/Fail Result
   31: EQU(Auto_Seq.Next_Step,190)MOV(200,Auto_Seq.Current_Step);
